// TIA Portal V19 export
TYPE "LAF_typeJobPrevious"
TITLE = LAF_typeMonitoring
// function block to select the job the EM should execute
// stored: Access Published
   STRUCT
      job { ExternalWritable := 'False'} : DInt;   // State number
      duration { ExternalWritable := 'False'} : LReal;   // Time stayed in that state
   END_STRUCT;
END_TYPE
